# EPICS substitutions: TEKMSO58LPApp/Db/mso58lp.substitutions
file dev_msoxx.template
{
    pattern {P,     PORT, NELM}
    {$(P),$(PORT),10000}
}

file "channel.template"
{
    pattern {P,     PORT,     CHANNEL,SCANTIME, NELM }
            {$(P),  $(PORT), 1,     "1 second",    10000}
            {$(P),  $(PORT), 2,     "1 second",    10000}
            {$(P),  $(PORT), 3,     "1 second",    10000}
            {$(P),  $(PORT), 4,     "1 second",    10000}
            {$(P),  $(PORT), 5,     "1 second",    10000}
            {$(P),  $(PORT), 6,     "1 second",    10000}
            {$(P),  $(PORT), 7,     "1 second",    10000}
            {$(P),  $(PORT), 8,     "1 second",    10000}
}
